{attribute 'qualified_only'}
{attribute 'strict'}
TYPE E_Barrier :
(
	eDisabled 			:= 0,	
	eError				:= 1,				// Stan nieaktywnosci (Stacja wyłączona)             
	eReady				:= 2,				// Stan gotowści do ruchu
	eWaitingToClose		:= 20,				// Stan oczekiwania na zamknięcie ( 1 faza, 4 wagi)
	eWaitingToOpen		:= 21,				// Stan oczekiwania na otwaricie ( 1 faza, 2 wagi)
	eClose				:= 30,				// Stan zamykania
	eOpen				:= 40,				// Stan otwarcia
	eDone				:= 50				// Wykonano cykl 
):=eDisabled;
END_TYPE

(* stored: Version 1.1.0.1, ProductVersion 3.1.4026.13, FileIdentifier 3a0bd165f9f6dc983d077b76223b2e8eb2293a58, FileSignature 716c15d874e413813735f9e64d5e037081aec41c801c80159d017851ba8c2fca87509ba2230a2e5d145b5865ed7fc624317dcf1874f757c97cfb4e2ef72a67ea1e0b7bd6179373c639fec0655d0f3e3ce98d5ac0a9151548e49e312cdf99addf41aa6ffb1f93d21888622f47af6447cf6df79491d19fbb06efc80f894f544598938650f27a84d644ff42b3ac9eec005f4052a2089157bcdee17c6a72f2e222e351ebdbb15a7ec5619f71f2ed973623a48ef729be9434420f3ee2309d9ea97951bd1cee91f2e780ff41472999b1cc8bb3c33bfb2a0587dc0d73f0a46e002f256cef420b5d10e5d3674ddf8010ab892dc5fd243f87889ee0b99c0236db9955e1a9
   DUT E_Barrier: Id {9640215a-87c3-46a3-a945-4ecb9e201072} *)
